{attribute 'linkalways'} 
{attribute 'no_explicit_call' := 'This FB is a CLASS and must be accessed using methods or properties'}
{attribute 'enable_dynamic_creation'}
FUNCTION_BLOCK NodePreExecuteEvent EXTENDS Disposable IMPLEMENTS I_NodePreExecuteEvent
VAR
	_target : I_Node;
	_cancelExecute : BOOL;
END_VAR

METHOD PUBLIC Cancel
VAR_INPUT
END_VAR
_cancelExecute := true;
END_METHOD

PROPERTY PUBLIC ExecuteCancelled : BOOL
GET
ExecuteCancelled := _cancelExecute;
END_GET
END_PROPERTY

METHOD FB_init : BOOL
VAR_INPUT
	bInitRetains : BOOL; // if TRUE, the retain variables are initialized (warm start / cold start)
	bInCopyCode : BOOL;  // if TRUE, the instance afterwards gets moved into the copy code (online change)
	Target : I_Node;
END_VAR
_target := Target;
END_METHOD

METHOD PUBLIC Reinitialize
VAR_INPUT
	Target : I_Node;
END_VAR
_cancelExecute := FALSE;
_target := Target;
END_METHOD

PROPERTY PUBLIC Target : I_Node
GET
Target := _target;
END_GET
END_PROPERTY

END_FUNCTION_BLOCK

(* stored: Version 1.1.0.1, ProductVersion 3.1.4024.13
   POU NodePreExecuteEvent: Id {6e27cc1e-c310-4d8f-82e7-28ae5f2b4bcc}, SpecialFunc None
   Folder Constructor: Id {37a2a32f-692b-4522-9061-94c8a73fda6b}
   Method Cancel: Id {4ecc4130-de8c-401d-be86-7c4cb9c56018}
   Property ExecuteCancelled: Id {b1cff844-64e2-4c8d-b97a-7f3dd22674c9}
   Get Get: Id {76bfbcfc-624f-4966-8e63-b6455db25a58}
   Method FB_init: Id {221b5ca8-b208-4530-840a-bd932741ae81}
   Method Reinitialize: Id {f74bec14-fa04-0cac-3a60-0f5190f71efb}
   Property Target: Id {e8cc0ba3-4643-4d25-ba56-3a31b949649f}
   Get Get: Id {34197992-a339-4436-b9bd-28db7ebd404d} *)
